FUNCTION_BLOCK fb_DBWrite
VAR_INPUT
	DataStruct:ST_DataStruct;
	Table:String(50);
END_VAR
VAR_OUTPUT
	bReady:bool:=false;
END_VAR
VAR
	bExecute:BOOL:=FALSE;
	
END_VAR

METHOD execute : BOOL
VAR_INPUT
END_VAR
bExecute:=TRUE;
END_METHOD

METHOD reset : BOOL
VAR_INPUT
END_VAR
bExecute:=FALSE;
bReady:=false;
END_METHOD

END_FUNCTION_BLOCK

(* stored: Version 1.1.0.1, ProductVersion 3.1.4024.2
   POU fb_DBWrite: Id {f338848e-13af-4a78-886c-9fcf7cd4df3a}, SpecialFunc None
   Method execute: Id {e5acd197-61d9-4ba5-ba7e-faad048654e0}
   Method reset: Id {5b328fe4-ef8d-4b13-9852-16fbc925a9a2} *)
